// TIA Portal project "Project_Metrou" (V15.1)

(* hardware
DEVICE "S71500/ET200MP station_1"  S7-1500 station
   slot 0: "Rail_0"  Rack  6ES7 590-1***0-0AA0
   slot 1: "PLC_1"  CPU 1513-1 PN  6ES7 513-1AL02-0AB0  V2.6
      slot 3: "CPU display_1"  6ES7591-1AA00-0AA0
DEVICE "HMI_1"  KTP900 Basic PN
   slot 0: "HMI_1"  KTP900 Basic PN  6AV2 123-2JB03-0AX0  15.1.0.0
   slot 1: "HMI_RT_1"  KTP900 Basic PN  6AV2 123-2JB03-0AX0  15.1.0.0
   slot 5: "HMI_1.IE_CP_1"  PROFINET Interface  15.0.1.0
      slot 1: "PROFINET Interface_1"  PROFINET Interface
         slot 1: "Port_1"  Port
*)

// ===== PLC "PLC_1"  CPU 1513-1 PN =====

DATA_BLOCK "Alarme_scara"   // DB1
{ S7_Optimized_Access := 'TRUE' }
VERSION : 0.1
   VAR
      alarme_gather : Word;
      alarme_vect : Array[0..15] of Bool;
   END_VAR
BEGIN
END_DATA_BLOCK

DATA_BLOCK "Avarii"   // DB2
{ S7_Optimized_Access := 'TRUE' }
VERSION : 0.1
   VAR
      esd : Bool;
      esd_btn : Bool;
      reset_esd : Bool;
      avarie_s1 : Bool;
      avarie_s2 : Bool;
      avarie_p1 : Bool;
      avarie_p2 : Bool;
      reset_avarii : Bool;
   END_VAR
BEGIN
END_DATA_BLOCK

DATA_BLOCK "Alarme_poarta"   // DB3
{ S7_Optimized_Access := 'TRUE' }
VERSION : 0.1
   VAR
      alarme_gather : Word;
      alarme_vect : Array[0..15] of Bool;
   END_VAR
BEGIN
END_DATA_BLOCK

DATA_BLOCK "Scara1_DB"   // DB4
{ S7_Optimized_Access := 'TRUE' }
VERSION : 0.1
// stored: InstanceOfName Scara
"Scara"
BEGIN
END_DATA_BLOCK

DATA_BLOCK "Scara2_DB"   // DB5
{ S7_Optimized_Access := 'TRUE' }
VERSION : 0.1
// stored: InstanceOfName Scara
"Scara"
BEGIN
END_DATA_BLOCK

DATA_BLOCK "Variabile_scara1"   // DB6
{ S7_Optimized_Access := 'TRUE' }
VERSION : 0.1
   VAR
      curent_stea : Real;
      curent_triunghi : Real;
      senzor_presiune : Bool;
      porniire_stea : Bool;
      pornire_triunghi : Bool;
      start : Bool;
      stop : Bool;
      directie : Bool;
      sus : Bool;
      jos : Bool;
      reseteaza_directia : Bool;
      start_sus : Bool;
      start_jos : Bool;
      cartela_intr : Bool;
   END_VAR
BEGIN
END_DATA_BLOCK

DATA_BLOCK "Variabile_scara2"   // DB7
{ S7_Optimized_Access := 'TRUE' }
VERSION : 0.1
   VAR
      curent_stea : Real;
      curent_triunghi : Real;
      senzor_presiune : Bool;
      porniire_stea : Bool;
      pornire_triunghi : Bool;
      start : Bool;
      stop : Bool;
      directie : Bool;
      sus : Bool;
      jos : Bool;
      reseteaza_directia : Bool;
      start_sus : Bool;
      start_jos : Bool;
      cartela_intr : Bool;
   END_VAR
BEGIN
END_DATA_BLOCK

DATA_BLOCK "Poarta1_DB"   // DB9
{ S7_Optimized_Access := 'TRUE' }
VERSION : 0.1
// stored: InstanceOfName Poarta
"Poarta"
BEGIN
END_DATA_BLOCK

DATA_BLOCK "Poarta2_DB"   // DB10
{ S7_Optimized_Access := 'TRUE' }
VERSION : 0.1
// stored: InstanceOfName Poarta
"Poarta"
BEGIN
END_DATA_BLOCK

DATA_BLOCK "Variabile_poarta1"   // DB11
{ S7_Optimized_Access := 'TRUE' }
VERSION : 0.1
   VAR
      cartela : Bool;
      stop : Bool;
      start : Bool;
      permisiune_start : Bool;
      start_intrare : Bool;
      start_iesire : Bool;
      s1 : Bool;
      s2 : Bool;
      p_deschis : Bool;
      alarma : Bool;
   END_VAR
BEGIN
END_DATA_BLOCK

DATA_BLOCK "Variabile_poarta2"   // DB12
{ S7_Optimized_Access := 'TRUE' }
VERSION : 0.1
   VAR
      cartela : Bool;
      stop : Bool;
      start : Bool;
      permisiune_start : Bool;
      start_intrare : Bool;
      start_iesire : Bool;
      s1 : Bool;
      s2 : Bool;
      p_deschis : Bool;
      alarma : Bool;
   END_VAR
BEGIN
END_DATA_BLOCK

// folder: System blocks/Program resources

DATA_BLOCK "reset_esd"   // DB8
{ S7_Optimized_Access := 'TRUE' }
AUTHOR : Simatic
FAMILY : IEC
NAME : IEC_TMR
VERSION : 1.0
// stored: InstanceOfName IEC_TIMER
"IEC_TIMER"
BEGIN
END_DATA_BLOCK

// folder: (top level)

FUNCTION_BLOCK "Scara"   // FB1, LAD
{ S7_Optimized_Access := 'TRUE' }
VERSION : 0.1
   VAR_INPUT
      esd : Bool;
      curent_stea : Real;
      curent_triunghi : Real;
      avarie_scara : Bool;
   END_VAR
   VAR_OUTPUT
      stea : Bool;
      triunghi : Bool;
   END_VAR
   VAR_IN_OUT
      senzor_presiune : Bool;
      reseteaza_directia : Bool;
      stop : Bool;
      start : Bool;
      start_sus : Bool;
      start_jos : Bool;
   END_VAR
   VAR
      sus : Bool;
      jos : Bool;
      pornire_stea : Bool;
      pornire_triunghi : Bool;
      permisiune_pornire : Bool;
      permisie_repornire : Bool;
      timer_stop : TON_TIME;
      Motor : "Motor";
   END_VAR
BEGIN

REGION Network 1: da permisiuneade pornire la scara
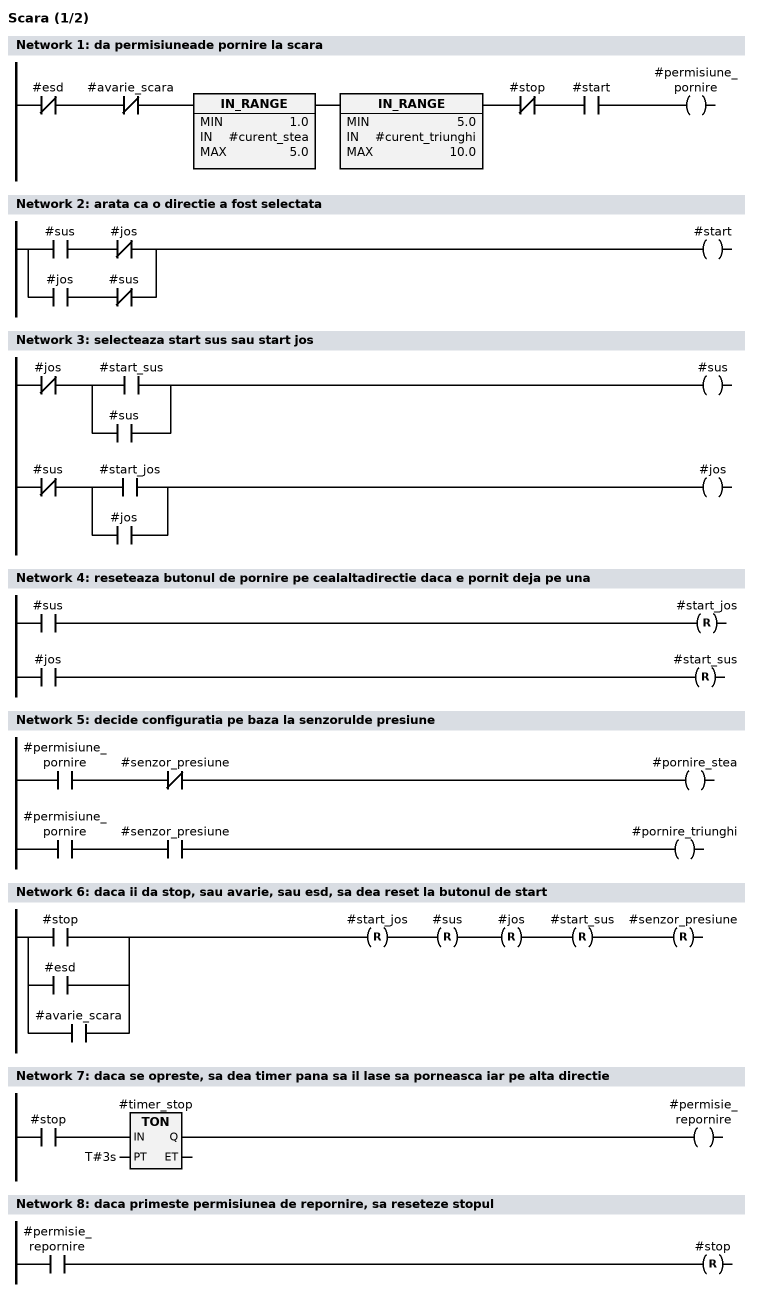
   RUNG wire#powerrail
      I_Contact( #esd )
      I_Contact( #avarie_scara )
      { S7_Templates := "SrcType := Real" } InRange(min := 1.0, in := #curent_stea, max := 5.0)
      { S7_Templates := "SrcType := Real" } InRange(min := 5.0, in := #curent_triunghi, max := 10.0)
      I_Contact( #stop )
      Contact( #start )
      Coil( #permisiune_pornire )
   END_RUNG
   // the same network as SCL:
   #permisiune_pornire := NOT #esd AND NOT #avarie_scara AND (1.0 <= #curent_stea) AND (#curent_stea <= 5.0) AND (5.0 <= #curent_triunghi) AND (#curent_triunghi <= 10.0) AND NOT #stop AND #start;
END_REGION

REGION Network 2: arata ca o directie a fost selectata
   RUNG wire#powerrail
      Contact( #sus )
      I_Contact( #jos )
      wire#w1
      Coil( #start )
   END_RUNG
   RUNG wire#powerrail
      Contact( #jos )
      I_Contact( #sus )
   END_RUNG wire#w1
   // the same network as SCL:
   #start := (#sus AND NOT #jos) OR (#jos AND NOT #sus);
END_REGION

REGION Network 3: selecteaza start sus sau start jos
   RUNG wire#powerrail
      I_Contact( #jos )
      wire#w1
      Contact( #start_sus )
      wire#w2
      Coil( #sus )
   END_RUNG
   RUNG wire#w1
      Contact( #sus )
   END_RUNG wire#w2
   RUNG wire#powerrail
      I_Contact( #sus )
      wire#w3
      Contact( #start_jos )
      wire#w4
      Coil( #jos )
   END_RUNG
   RUNG wire#w3
      Contact( #jos )
   END_RUNG wire#w4
   // the same network as SCL:
   #sus := NOT #jos AND (#start_sus OR #sus);
   #jos := NOT #sus AND (#start_jos OR #jos);
END_REGION

REGION Network 4: reseteaza butonul de pornire pe cealaltadirectie daca e pornit deja pe una
   RUNG wire#powerrail
      Contact( #sus )
      R_Coil( #start_jos )
   END_RUNG
   RUNG wire#powerrail
      Contact( #jos )
      R_Coil( #start_sus )
   END_RUNG
   // the same network as SCL:
   IF #sus THEN #start_jos := FALSE; END_IF;
   IF #jos THEN #start_sus := FALSE; END_IF;
END_REGION

REGION Network 5: decide configuratia pe baza la senzorulde presiune
   RUNG wire#powerrail
      Contact( #permisiune_pornire )
      I_Contact( #senzor_presiune )
      Coil( #pornire_stea )
   END_RUNG
   RUNG wire#powerrail
      Contact( #permisiune_pornire )
      Contact( #senzor_presiune )
      Coil( #pornire_triunghi )
   END_RUNG
   // the same network as SCL:
   #pornire_stea := #permisiune_pornire AND NOT #senzor_presiune;
   #pornire_triunghi := #permisiune_pornire AND #senzor_presiune;
END_REGION

REGION Network 6: daca ii da stop, sau avarie, sau esd, sa dea reset la butonul de start
   RUNG wire#powerrail
      Contact( #stop )
      wire#w1
      R_Coil( #start_jos )
      R_Coil( #sus )
      R_Coil( #jos )
      R_Coil( #start_sus )
      R_Coil( #senzor_presiune )
   END_RUNG
   RUNG wire#powerrail
      Contact( #esd )
   END_RUNG wire#w1
   RUNG wire#powerrail
      Contact( #avarie_scara )
   END_RUNG wire#w1
   // the same network as SCL:
   IF #stop OR #esd OR #avarie_scara THEN
       #start_jos := FALSE;
       #sus := FALSE;
       #jos := FALSE;
       #start_sus := FALSE;
       #senzor_presiune := FALSE;
   END_IF;
END_REGION

REGION Network 7: daca se opreste, sa dea timer pana sa il lase sa porneasca iar pe alta directie
   #timer_stop(IN := #stop, PT := T#3s);   // TON
   #permisie_repornire := #timer_stop.Q;
END_REGION

REGION Network 8: daca primeste permisiunea de repornire, sa reseteze stopul
   RUNG wire#powerrail
      Contact( #permisie_repornire )
      R_Coil( #stop )
   END_RUNG
   // the same network as SCL:
   IF #permisie_repornire THEN #stop := FALSE; END_IF;
END_REGION

REGION Network 9: functia de motor a scarii
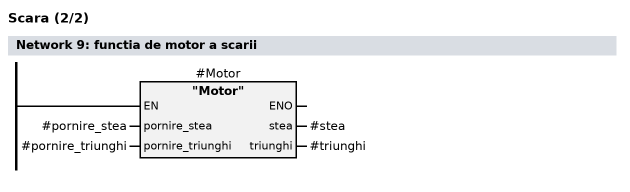
   RUNG wire#powerrail
      #Motor(pornire_stea := #pornire_stea, pornire_triunghi := #pornire_triunghi, stea => #stea, triunghi => #triunghi)
   END_RUNG
   // the same network as SCL:
   #Motor(pornire_stea := #pornire_stea,   // "Motor"
          pornire_triunghi := #pornire_triunghi,
          stea => #stea,
          triunghi => #triunghi);
END_REGION
END_FUNCTION_BLOCK

FUNCTION_BLOCK "Motor"   // FB2, LAD
{ S7_Optimized_Access := 'TRUE' }
VERSION : 0.1
   VAR_INPUT
      pornire_stea : Bool;
      pornire_triunghi : Bool;
   END_VAR
   VAR_OUTPUT
      stea : Bool;
      triunghi : Bool;
   END_VAR
BEGIN

REGION Network 1: daca primeste plecare pe stea, sa o activeze
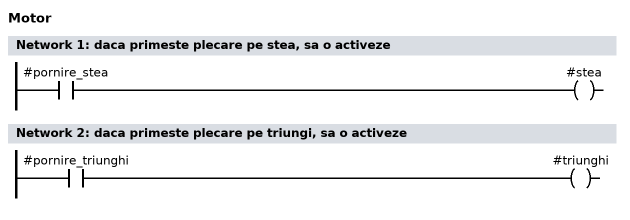
   RUNG wire#powerrail
      Contact( #pornire_stea )
      Coil( #stea )
   END_RUNG
   // the same network as SCL:
   #stea := #pornire_stea;
END_REGION

REGION Network 2: daca primeste plecare pe triungi, sa o activeze
   RUNG wire#powerrail
      Contact( #pornire_triunghi )
      Coil( #triunghi )
   END_RUNG
   // the same network as SCL:
   #triunghi := #pornire_triunghi;
END_REGION
END_FUNCTION_BLOCK

FUNCTION_BLOCK "Poarta"   // FB3, LAD
{ S7_Optimized_Access := 'TRUE' }
VERSION : 0.1
   VAR_INPUT
      esd : Bool;
      avarie_poarta : Bool;
   END_VAR
   VAR_OUTPUT
      poarta_deschisa : Bool;
      alarma : Bool;
   END_VAR
   VAR_IN_OUT
      senzor1 : Bool;
      senzor2 : Bool;
      cartela : Bool;
      stop : Bool;
      start : Bool;
      permisiune_start : Bool;
      start_intrare : Bool;
      start_iesire : Bool;
      cartela_introdusa : Bool;
   END_VAR
   VAR
      terminat1 : Bool;
      terminat2 : Bool;
      intrare : Bool;
      s1_intrare : Bool;
      s1_iesire : Bool;
      s2_intrare : Bool;
      s2_iesire : Bool;
      iesire : Bool;
      reset_stop : TON_TIME;
      Iesire_metrou_Instance : "Iesire_metrou";
      Intrare_metrou_Instance : "Intrare_metrou";
   END_VAR
BEGIN

REGION Network 1: porneste poarta
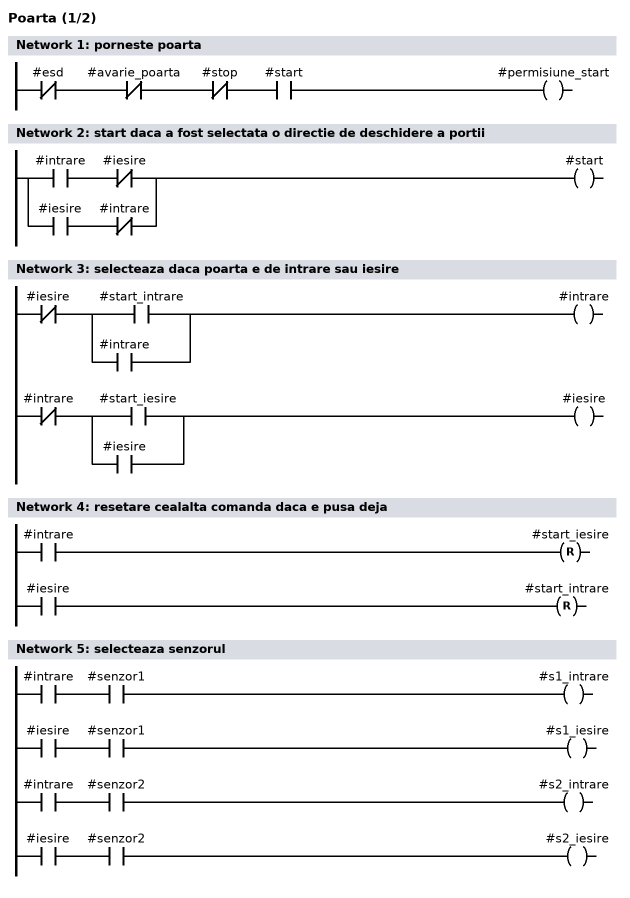
   RUNG wire#powerrail
      I_Contact( #esd )
      I_Contact( #avarie_poarta )
      I_Contact( #stop )
      Contact( #start )
      Coil( #permisiune_start )
   END_RUNG
   // the same network as SCL:
   #permisiune_start := NOT #esd AND NOT #avarie_poarta AND NOT #stop AND #start;
END_REGION

REGION Network 2: start daca a fost selectata o directie de deschidere a portii
   RUNG wire#powerrail
      Contact( #intrare )
      I_Contact( #iesire )
      wire#w1
      Coil( #start )
   END_RUNG
   RUNG wire#powerrail
      Contact( #iesire )
      I_Contact( #intrare )
   END_RUNG wire#w1
   // the same network as SCL:
   #start := (#intrare AND NOT #iesire) OR (#iesire AND NOT #intrare);
END_REGION

REGION Network 3: selecteaza daca poarta e de intrare sau iesire
   RUNG wire#powerrail
      I_Contact( #iesire )
      wire#w1
      Contact( #start_intrare )
      wire#w2
      Coil( #intrare )
   END_RUNG
   RUNG wire#w1
      Contact( #intrare )
   END_RUNG wire#w2
   RUNG wire#powerrail
      I_Contact( #intrare )
      wire#w3
      Contact( #start_iesire )
      wire#w4
      Coil( #iesire )
   END_RUNG
   RUNG wire#w3
      Contact( #iesire )
   END_RUNG wire#w4
   // the same network as SCL:
   #intrare := NOT #iesire AND (#start_intrare OR #intrare);
   #iesire := NOT #intrare AND (#start_iesire OR #iesire);
END_REGION

REGION Network 4: resetare cealalta comanda daca e pusa deja
   RUNG wire#powerrail
      Contact( #intrare )
      R_Coil( #start_iesire )
   END_RUNG
   RUNG wire#powerrail
      Contact( #iesire )
      R_Coil( #start_intrare )
   END_RUNG
   // the same network as SCL:
   IF #intrare THEN #start_iesire := FALSE; END_IF;
   IF #iesire THEN #start_intrare := FALSE; END_IF;
END_REGION

REGION Network 5: selecteaza senzorul
   RUNG wire#powerrail
      Contact( #intrare )
      Contact( #senzor1 )
      Coil( #s1_intrare )
   END_RUNG
   RUNG wire#powerrail
      Contact( #iesire )
      Contact( #senzor1 )
      Coil( #s1_iesire )
   END_RUNG
   RUNG wire#powerrail
      Contact( #intrare )
      Contact( #senzor2 )
      Coil( #s2_intrare )
   END_RUNG
   RUNG wire#powerrail
      Contact( #iesire )
      Contact( #senzor2 )
      Coil( #s2_iesire )
   END_RUNG
   // the same network as SCL:
   #s1_intrare := #intrare AND #senzor1;
   #s1_iesire := #iesire AND #senzor1;
   #s2_intrare := #intrare AND #senzor2;
   #s2_iesire := #iesire AND #senzor2;
END_REGION

REGION Network 6: functie intrare/iesire
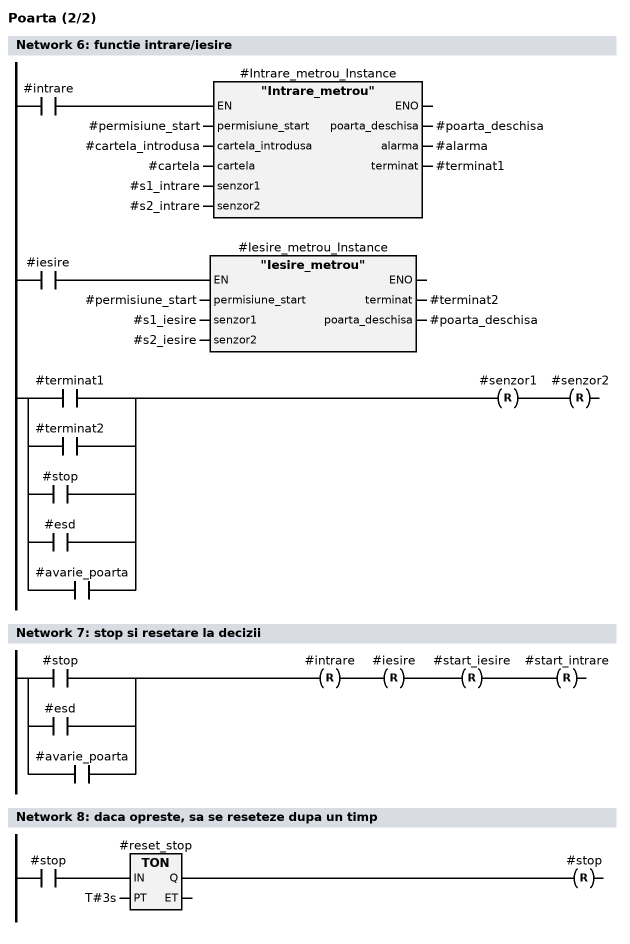
   RUNG wire#powerrail
      Contact( #intrare )
      #Intrare_metrou_Instance(permisiune_start := #permisiune_start, cartela_introdusa := #cartela_introdusa, cartela := #cartela, senzor1 := #s1_intrare, senzor2 := #s2_intrare, poarta_deschisa => #poarta_deschisa, alarma => #alarma, terminat => #terminat1)
   END_RUNG
   RUNG wire#powerrail
      Contact( #iesire )
      #Iesire_metrou_Instance(permisiune_start := #permisiune_start, senzor1 := #s1_iesire, senzor2 := #s2_iesire, terminat => #terminat2, poarta_deschisa => #poarta_deschisa)
   END_RUNG
   RUNG wire#powerrail
      Contact( #terminat1 )
      wire#w1
      R_Coil( #senzor1 )
      R_Coil( #senzor2 )
   END_RUNG
   RUNG wire#powerrail
      Contact( #terminat2 )
   END_RUNG wire#w1
   RUNG wire#powerrail
      Contact( #stop )
   END_RUNG wire#w1
   RUNG wire#powerrail
      Contact( #esd )
   END_RUNG wire#w1
   RUNG wire#powerrail
      Contact( #avarie_poarta )
   END_RUNG wire#w1
   // the same network as SCL:
   IF #intrare THEN
       #Intrare_metrou_Instance(permisiune_start := #permisiune_start,   // "Intrare_metrou"
                               cartela_introdusa := #cartela_introdusa,
                               cartela := #cartela,
                               senzor1 := #s1_intrare,
                               senzor2 := #s2_intrare,
                               poarta_deschisa => #poarta_deschisa,
                               alarma => #alarma,
                               terminat => #terminat1);
   END_IF;
   IF #iesire THEN
       #Iesire_metrou_Instance(permisiune_start := #permisiune_start,   // "Iesire_metrou"
                               senzor1 := #s1_iesire,
                               senzor2 := #s2_iesire,
                               terminat => #terminat2,
                               poarta_deschisa => #poarta_deschisa);
   END_IF;
   IF #terminat1 OR #terminat2 OR #stop OR #esd OR #avarie_poarta THEN
       #senzor1 := FALSE;
       #senzor2 := FALSE;
   END_IF;
END_REGION

REGION Network 7: stop si resetare la decizii
   RUNG wire#powerrail
      Contact( #stop )
      wire#w1
      R_Coil( #intrare )
      R_Coil( #iesire )
      R_Coil( #start_iesire )
      R_Coil( #start_intrare )
   END_RUNG
   RUNG wire#powerrail
      Contact( #esd )
   END_RUNG wire#w1
   RUNG wire#powerrail
      Contact( #avarie_poarta )
   END_RUNG wire#w1
   // the same network as SCL:
   IF #stop OR #esd OR #avarie_poarta THEN
       #intrare := FALSE;
       #iesire := FALSE;
       #start_iesire := FALSE;
       #start_intrare := FALSE;
   END_IF;
END_REGION

REGION Network 8: daca opreste, sa se reseteze dupa un timp
   #reset_stop(IN := #stop, PT := T#3s);   // TON
   IF #reset_stop.Q THEN #stop := FALSE; END_IF;
END_REGION
END_FUNCTION_BLOCK

FUNCTION_BLOCK "Intrare_metrou"   // FB4, LAD
{ S7_Optimized_Access := 'TRUE' }
VERSION : 0.1
   VAR_INPUT
      permisiune_start : Bool;
   END_VAR
   VAR_OUTPUT
      poarta_deschisa : Bool;
      alarma : Bool;
      terminat : Bool;
   END_VAR
   VAR_IN_OUT
      cartela_introdusa : Bool;
      cartela : Bool;
      senzor1 : Bool;
      senzor2 : Bool;
   END_VAR
   VAR
      timer_alarma : TON_TIME;
   END_VAR
BEGIN

REGION Network 1
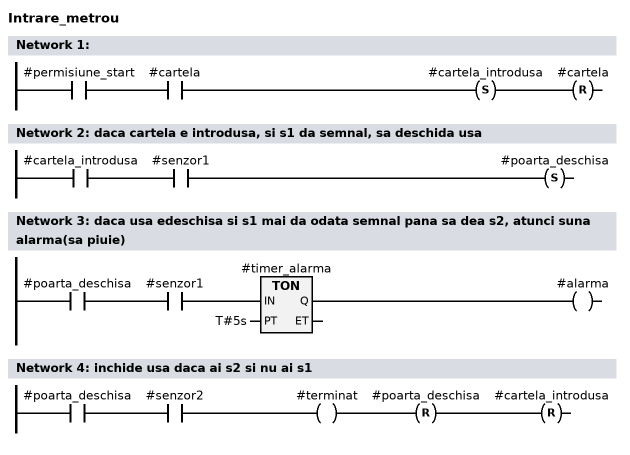
   RUNG wire#powerrail
      Contact( #permisiune_start )
      Contact( #cartela )
      S_Coil( #cartela_introdusa )
      R_Coil( #cartela )
   END_RUNG
   // the same network as SCL:
   IF #permisiune_start AND #cartela THEN
       #cartela_introdusa := TRUE;
       #cartela := FALSE;
   END_IF;
END_REGION

REGION Network 2: daca cartela e introdusa, si s1 da semnal, sa deschida usa
   RUNG wire#powerrail
      Contact( #cartela_introdusa )
      Contact( #senzor1 )
      S_Coil( #poarta_deschisa )
   END_RUNG
   // the same network as SCL:
   IF #cartela_introdusa AND #senzor1 THEN #poarta_deschisa := TRUE; END_IF;
END_REGION

REGION Network 3: daca usa edeschisa si s1 mai da odata semnal pana sa dea s2, atunci suna alarma(sa piuie)
   #timer_alarma(IN := #poarta_deschisa AND #senzor1, PT := T#5s);   // TON
   #alarma := #timer_alarma.Q;
END_REGION

REGION Network 4: inchide usa daca ai s2 si nu ai s1
   RUNG wire#powerrail
      Contact( #poarta_deschisa )
      Contact( #senzor2 )
      Coil( #terminat )
      R_Coil( #poarta_deschisa )
      R_Coil( #cartela_introdusa )
   END_RUNG
   // the same network as SCL:
   #terminat := #poarta_deschisa AND #senzor2;
   IF #terminat THEN
       #poarta_deschisa := FALSE;
       #cartela_introdusa := FALSE;
   END_IF;
END_REGION
END_FUNCTION_BLOCK

FUNCTION_BLOCK "Iesire_metrou"   // FB5, LAD
{ S7_Optimized_Access := 'TRUE' }
VERSION : 0.1
   VAR_INPUT
      permisiune_start : Bool;
   END_VAR
   VAR_OUTPUT
      terminat : Bool;
      poarta_deschisa : Bool;
   END_VAR
   VAR_IN_OUT
      senzor1 : Bool;
      senzor2 : Bool;
   END_VAR
BEGIN

REGION Network 1: deschide poarta daca senzor1 da semnal
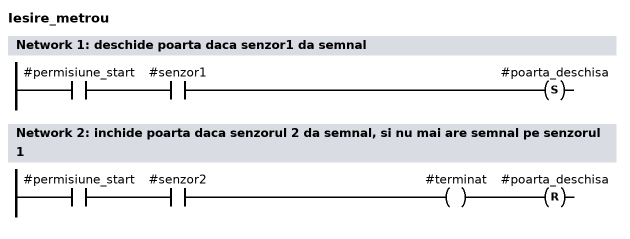
   RUNG wire#powerrail
      Contact( #permisiune_start )
      Contact( #senzor1 )
      S_Coil( #poarta_deschisa )
   END_RUNG
   // the same network as SCL:
   IF #permisiune_start AND #senzor1 THEN #poarta_deschisa := TRUE; END_IF;
END_REGION

REGION Network 2: inchide poarta daca senzorul 2 da semnal, si nu mai are semnal pe senzorul 1
   RUNG wire#powerrail
      Contact( #permisiune_start )
      Contact( #senzor2 )
      Coil( #terminat )
      R_Coil( #poarta_deschisa )
   END_RUNG
   // the same network as SCL:
   #terminat := #permisiune_start AND #senzor2;
   IF #terminat THEN #poarta_deschisa := FALSE; END_IF;
END_REGION
END_FUNCTION_BLOCK

ORGANIZATION_BLOCK "Main"   // OB1, LAD, ProgramCycle
TITLE = "Main Program Sweep (Cycle)"
{ S7_Optimized_Access := 'TRUE' }
VERSION : 0.1
   VAR_INPUT
      Initial_Call : Bool;   // Initial call of this OB
      Remanence : Bool;   // =True, if remanent data are available
   END_VAR
   VAR_TEMP   // added for the SCL form of the ladder/FBD networks
      _w1 : Bool;
      _w2 : Bool;
      _w3 : Bool;
      _w4 : Bool;
   END_VAR
BEGIN

REGION Network 1: scara 1
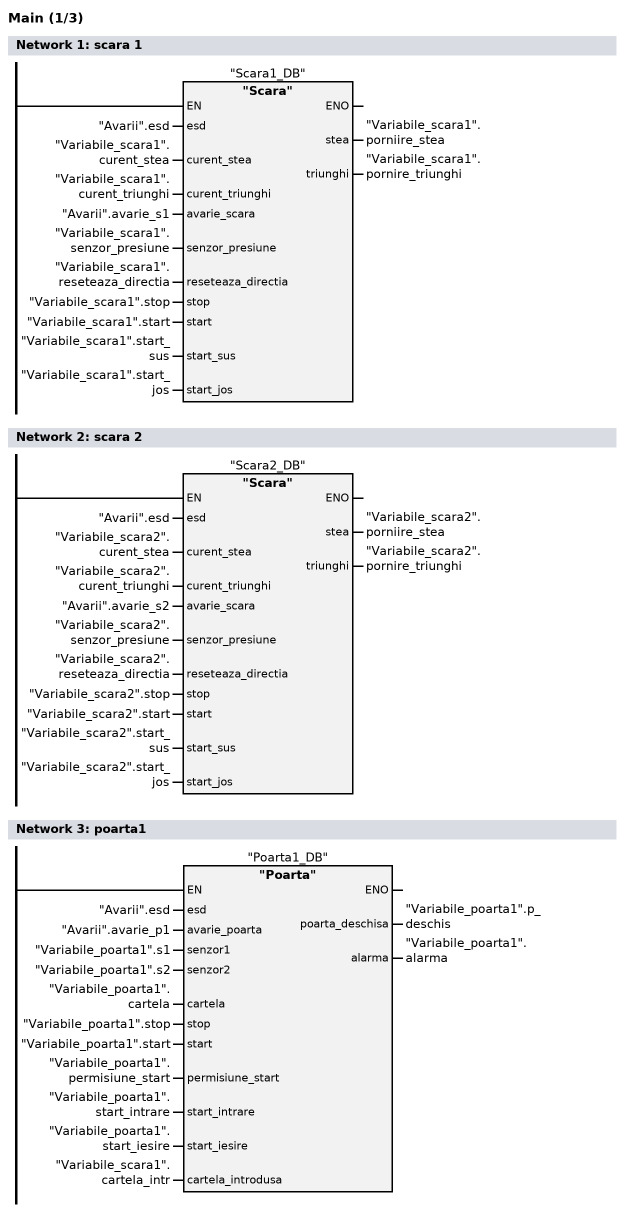
   RUNG wire#powerrail
      "Scara1_DB"(esd := "Avarii".esd, curent_stea := "Variabile_scara1".curent_stea, curent_triunghi := "Variabile_scara1".curent_triunghi, avarie_scara := "Avarii".avarie_s1, senzor_presiune := "Variabile_scara1".senzor_presiune, reseteaza_directia := "Variabile_scara1".reseteaza_directia, stop := "Variabile_scara1".stop, start := "Variabile_scara1".start, start_sus := "Variabile_scara1".start_sus, start_jos := "Variabile_scara1".start_jos, stea => "Variabile_scara1".porniire_stea, triunghi => "Variabile_scara1".pornire_triunghi)
   END_RUNG
   // the same network as SCL:
   "Scara1_DB"(esd := "Avarii".esd,   // "Scara"
               curent_stea := "Variabile_scara1".curent_stea,
               curent_triunghi := "Variabile_scara1".curent_triunghi,
               avarie_scara := "Avarii".avarie_s1,
               senzor_presiune := "Variabile_scara1".senzor_presiune,
               reseteaza_directia := "Variabile_scara1".reseteaza_directia,
               stop := "Variabile_scara1".stop,
               start := "Variabile_scara1".start,
               start_sus := "Variabile_scara1".start_sus,
               start_jos := "Variabile_scara1".start_jos,
               stea => "Variabile_scara1".porniire_stea,
               triunghi => "Variabile_scara1".pornire_triunghi);
END_REGION

REGION Network 2: scara 2
   RUNG wire#powerrail
      "Scara2_DB"(esd := "Avarii".esd, curent_stea := "Variabile_scara2".curent_stea, curent_triunghi := "Variabile_scara2".curent_triunghi, avarie_scara := "Avarii".avarie_s2, senzor_presiune := "Variabile_scara2".senzor_presiune, reseteaza_directia := "Variabile_scara2".reseteaza_directia, stop := "Variabile_scara2".stop, start := "Variabile_scara2".start, start_sus := "Variabile_scara2".start_sus, start_jos := "Variabile_scara2".start_jos, stea => "Variabile_scara2".porniire_stea, triunghi => "Variabile_scara2".pornire_triunghi)
   END_RUNG
   // the same network as SCL:
   "Scara2_DB"(esd := "Avarii".esd,   // "Scara"
               curent_stea := "Variabile_scara2".curent_stea,
               curent_triunghi := "Variabile_scara2".curent_triunghi,
               avarie_scara := "Avarii".avarie_s2,
               senzor_presiune := "Variabile_scara2".senzor_presiune,
               reseteaza_directia := "Variabile_scara2".reseteaza_directia,
               stop := "Variabile_scara2".stop,
               start := "Variabile_scara2".start,
               start_sus := "Variabile_scara2".start_sus,
               start_jos := "Variabile_scara2".start_jos,
               stea => "Variabile_scara2".porniire_stea,
               triunghi => "Variabile_scara2".pornire_triunghi);
END_REGION

REGION Network 3: poarta1
   RUNG wire#powerrail
      "Poarta1_DB"(esd := "Avarii".esd, avarie_poarta := "Avarii".avarie_p1, senzor1 := "Variabile_poarta1".s1, senzor2 := "Variabile_poarta1".s2, cartela := "Variabile_poarta1".cartela, stop := "Variabile_poarta1".stop, start := "Variabile_poarta1".start, permisiune_start := "Variabile_poarta1".permisiune_start, start_intrare := "Variabile_poarta1".start_intrare, start_iesire := "Variabile_poarta1".start_iesire, cartela_introdusa := "Variabile_scara1".cartela_intr, poarta_deschisa => "Variabile_poarta1".p_deschis, alarma => "Variabile_poarta1".alarma)
   END_RUNG
   // the same network as SCL:
   "Poarta1_DB"(esd := "Avarii".esd,   // "Poarta"
                avarie_poarta := "Avarii".avarie_p1,
                senzor1 := "Variabile_poarta1".s1,
                senzor2 := "Variabile_poarta1".s2,
                cartela := "Variabile_poarta1".cartela,
                stop := "Variabile_poarta1".stop,
                start := "Variabile_poarta1".start,
                permisiune_start := "Variabile_poarta1".permisiune_start,
                start_intrare := "Variabile_poarta1".start_intrare,
                start_iesire := "Variabile_poarta1".start_iesire,
                cartela_introdusa := "Variabile_scara1".cartela_intr,
                poarta_deschisa => "Variabile_poarta1".p_deschis,
                alarma => "Variabile_poarta1".alarma);
END_REGION

REGION Network 4: poarta2
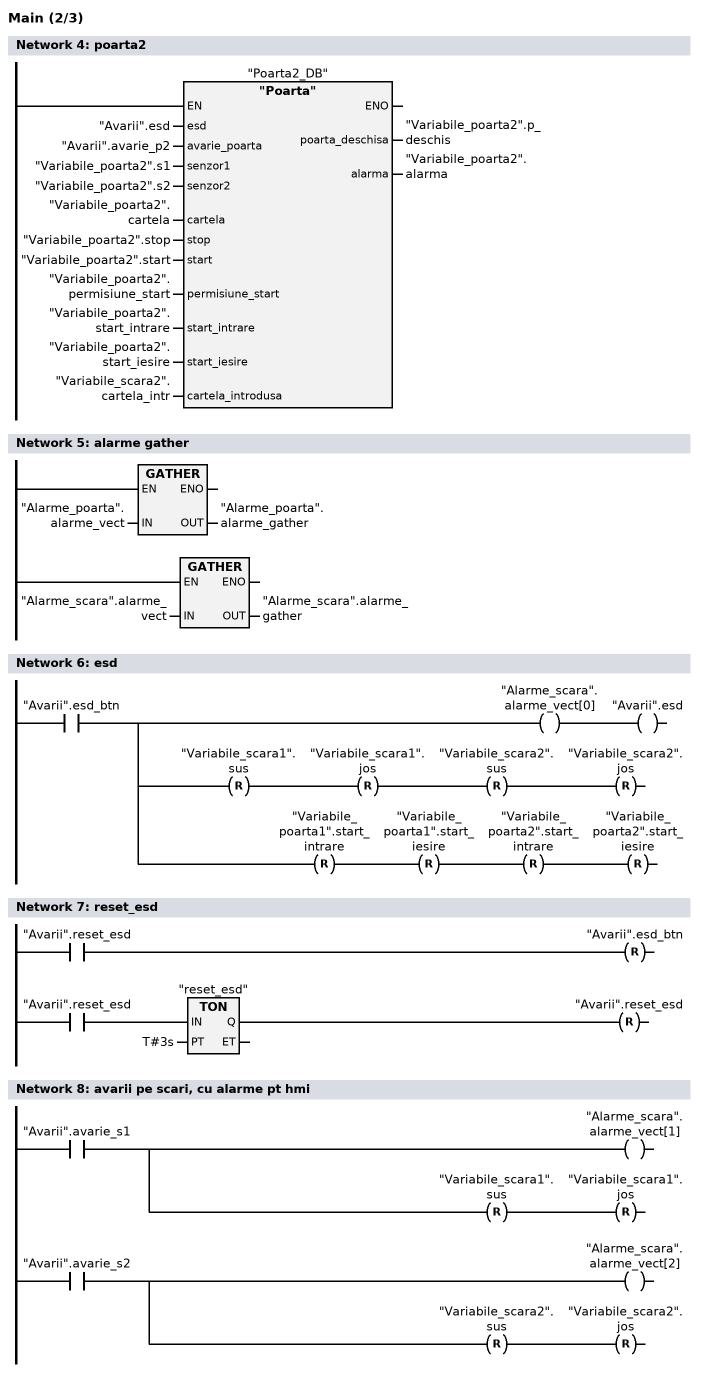
   RUNG wire#powerrail
      "Poarta2_DB"(esd := "Avarii".esd, avarie_poarta := "Avarii".avarie_p2, senzor1 := "Variabile_poarta2".s1, senzor2 := "Variabile_poarta2".s2, cartela := "Variabile_poarta2".cartela, stop := "Variabile_poarta2".stop, start := "Variabile_poarta2".start, permisiune_start := "Variabile_poarta2".permisiune_start, start_intrare := "Variabile_poarta2".start_intrare, start_iesire := "Variabile_poarta2".start_iesire, cartela_introdusa := "Variabile_scara2".cartela_intr, poarta_deschisa => "Variabile_poarta2".p_deschis, alarma => "Variabile_poarta2".alarma)
   END_RUNG
   // the same network as SCL:
   "Poarta2_DB"(esd := "Avarii".esd,   // "Poarta"
                avarie_poarta := "Avarii".avarie_p2,
                senzor1 := "Variabile_poarta2".s1,
                senzor2 := "Variabile_poarta2".s2,
                cartela := "Variabile_poarta2".cartela,
                stop := "Variabile_poarta2".stop,
                start := "Variabile_poarta2".start,
                permisiune_start := "Variabile_poarta2".permisiune_start,
                start_intrare := "Variabile_poarta2".start_intrare,
                start_iesire := "Variabile_poarta2".start_iesire,
                cartela_introdusa := "Variabile_scara2".cartela_intr,
                poarta_deschisa => "Variabile_poarta2".p_deschis,
                alarma => "Variabile_poarta2".alarma);
END_REGION

REGION Network 5: alarme gather
   GATHER(IN := "Alarme_poarta".alarme_vect, OUT => "Alarme_poarta".alarme_gather);
   GATHER(IN := "Alarme_scara".alarme_vect, OUT => "Alarme_scara".alarme_gather);
END_REGION

REGION Network 6: esd
   RUNG wire#powerrail
      Contact( "Avarii".esd_btn )
      wire#w1
      Coil( "Alarme_scara".alarme_vect[0] )
      Coil( "Avarii".esd )
   END_RUNG
   RUNG wire#w1
      R_Coil( "Variabile_scara1".sus )
      R_Coil( "Variabile_scara1".jos )
      R_Coil( "Variabile_scara2".sus )
      R_Coil( "Variabile_scara2".jos )
   END_RUNG
   RUNG wire#w1
      R_Coil( "Variabile_poarta1".start_intrare )
      R_Coil( "Variabile_poarta1".start_iesire )
      R_Coil( "Variabile_poarta2".start_intrare )
      R_Coil( "Variabile_poarta2".start_iesire )
   END_RUNG
   // the same network as SCL:
   "Alarme_scara".alarme_vect[0] := "Avarii".esd_btn;
   "Avarii".esd := "Avarii".esd_btn;
   IF "Avarii".esd_btn THEN
       "Variabile_scara1".sus := FALSE;
       "Variabile_scara1".jos := FALSE;
       "Variabile_scara2".sus := FALSE;
       "Variabile_scara2".jos := FALSE;
       "Variabile_poarta1".start_intrare := FALSE;
       "Variabile_poarta1".start_iesire := FALSE;
       "Variabile_poarta2".start_intrare := FALSE;
       "Variabile_poarta2".start_iesire := FALSE;
   END_IF;
END_REGION

REGION Network 7: reset_esd
   IF "Avarii".reset_esd THEN "Avarii".esd_btn := FALSE; END_IF;
   "reset_esd".TON(IN := "Avarii".reset_esd, PT := T#3s);
   IF "reset_esd".Q THEN "Avarii".reset_esd := FALSE; END_IF;
END_REGION

REGION Network 8: avarii pe scari, cu alarme pt hmi
   RUNG wire#powerrail
      Contact( "Avarii".avarie_s1 )
      wire#w1
      Coil( "Alarme_scara".alarme_vect[1] )
   END_RUNG
   RUNG wire#w1
      R_Coil( "Variabile_scara1".sus )
      R_Coil( "Variabile_scara1".jos )
   END_RUNG
   RUNG wire#powerrail
      Contact( "Avarii".avarie_s2 )
      wire#w2
      Coil( "Alarme_scara".alarme_vect[2] )
   END_RUNG
   RUNG wire#w2
      R_Coil( "Variabile_scara2".sus )
      R_Coil( "Variabile_scara2".jos )
   END_RUNG
   // the same network as SCL:
   "Alarme_scara".alarme_vect[1] := "Avarii".avarie_s1;
   IF "Avarii".avarie_s1 THEN
       "Variabile_scara1".sus := FALSE;
       "Variabile_scara1".jos := FALSE;
   END_IF;
   "Alarme_scara".alarme_vect[2] := "Avarii".avarie_s2;
   IF "Avarii".avarie_s2 THEN
       "Variabile_scara2".sus := FALSE;
       "Variabile_scara2".jos := FALSE;
   END_IF;
END_REGION

REGION Network 9: reset la avarii
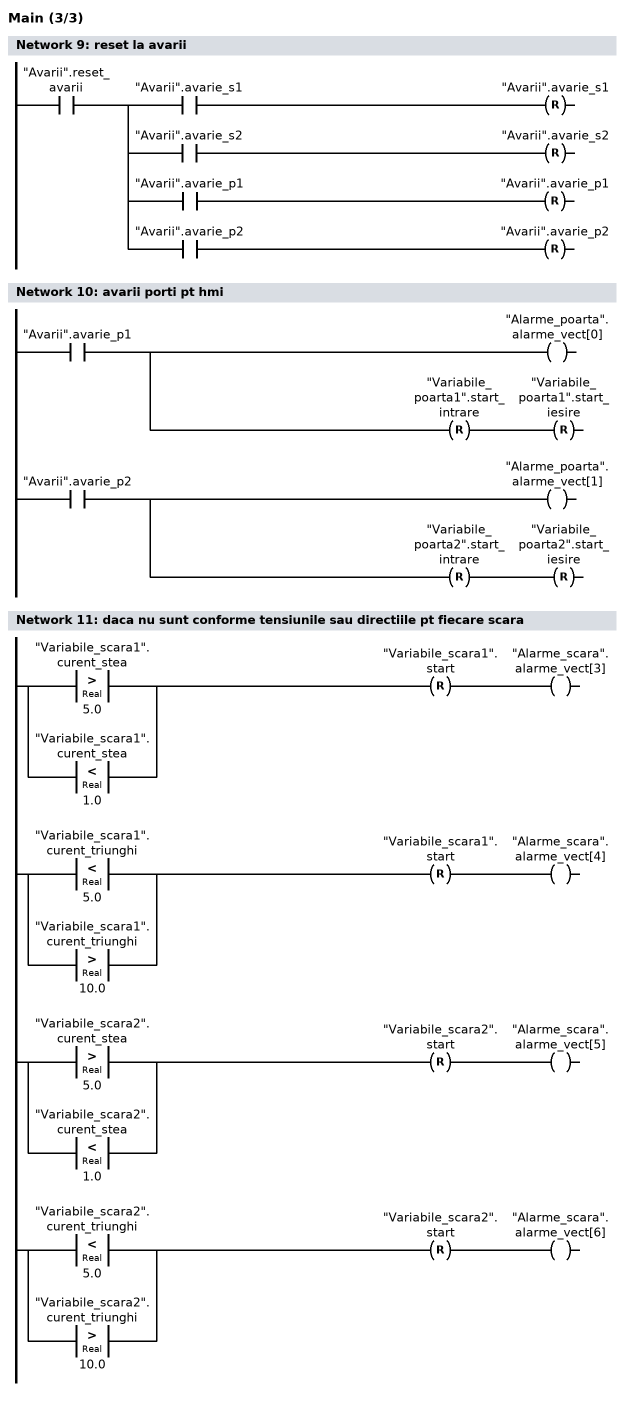
   RUNG wire#powerrail
      Contact( "Avarii".reset_avarii )
      wire#w1
      Contact( "Avarii".avarie_s1 )
      R_Coil( "Avarii".avarie_s1 )
   END_RUNG
   RUNG wire#w1
      Contact( "Avarii".avarie_s2 )
      R_Coil( "Avarii".avarie_s2 )
   END_RUNG
   RUNG wire#w1
      Contact( "Avarii".avarie_p1 )
      R_Coil( "Avarii".avarie_p1 )
   END_RUNG
   RUNG wire#w1
      Contact( "Avarii".avarie_p2 )
      R_Coil( "Avarii".avarie_p2 )
   END_RUNG
   // the same network as SCL:
   IF "Avarii".reset_avarii AND "Avarii".avarie_s1 THEN "Avarii".avarie_s1 := FALSE; END_IF;
   IF "Avarii".reset_avarii AND "Avarii".avarie_s2 THEN "Avarii".avarie_s2 := FALSE; END_IF;
   IF "Avarii".reset_avarii AND "Avarii".avarie_p1 THEN "Avarii".avarie_p1 := FALSE; END_IF;
   IF "Avarii".reset_avarii AND "Avarii".avarie_p2 THEN "Avarii".avarie_p2 := FALSE; END_IF;
END_REGION

REGION Network 10: avarii porti pt hmi
   RUNG wire#powerrail
      Contact( "Avarii".avarie_p1 )
      wire#w1
      Coil( "Alarme_poarta".alarme_vect[0] )
   END_RUNG
   RUNG wire#w1
      R_Coil( "Variabile_poarta1".start_intrare )
      R_Coil( "Variabile_poarta1".start_iesire )
   END_RUNG
   RUNG wire#powerrail
      Contact( "Avarii".avarie_p2 )
      wire#w2
      Coil( "Alarme_poarta".alarme_vect[1] )
   END_RUNG
   RUNG wire#w2
      R_Coil( "Variabile_poarta2".start_intrare )
      R_Coil( "Variabile_poarta2".start_iesire )
   END_RUNG
   // the same network as SCL:
   "Alarme_poarta".alarme_vect[0] := "Avarii".avarie_p1;
   IF "Avarii".avarie_p1 THEN
       "Variabile_poarta1".start_intrare := FALSE;
       "Variabile_poarta1".start_iesire := FALSE;
   END_IF;
   "Alarme_poarta".alarme_vect[1] := "Avarii".avarie_p2;
   IF "Avarii".avarie_p2 THEN
       "Variabile_poarta2".start_intrare := FALSE;
       "Variabile_poarta2".start_iesire := FALSE;
   END_IF;
END_REGION

REGION Network 11: daca nu sunt conforme tensiunile sau directiile pt fiecare scara
   RUNG wire#powerrail
      { S7_Templates := "SrcType := Real" } GT_Contact(in1 := "Variabile_scara1".curent_stea, in2 := 5.0)
      wire#w1
      R_Coil( "Variabile_scara1".start )
      Coil( "Alarme_scara".alarme_vect[3] )
   END_RUNG
   RUNG wire#powerrail
      { S7_Templates := "SrcType := Real" } LT_Contact(in1 := "Variabile_scara1".curent_stea, in2 := 1.0)
   END_RUNG wire#w1
   RUNG wire#powerrail
      { S7_Templates := "SrcType := Real" } LT_Contact(in1 := "Variabile_scara1".curent_triunghi, in2 := 5.0)
      wire#w2
      R_Coil( "Variabile_scara1".start )
      Coil( "Alarme_scara".alarme_vect[4] )
   END_RUNG
   RUNG wire#powerrail
      { S7_Templates := "SrcType := Real" } GT_Contact(in1 := "Variabile_scara1".curent_triunghi, in2 := 10.0)
   END_RUNG wire#w2
   RUNG wire#powerrail
      { S7_Templates := "SrcType := Real" } GT_Contact(in1 := "Variabile_scara2".curent_stea, in2 := 5.0)
      wire#w3
      R_Coil( "Variabile_scara2".start )
      Coil( "Alarme_scara".alarme_vect[5] )
   END_RUNG
   RUNG wire#powerrail
      { S7_Templates := "SrcType := Real" } LT_Contact(in1 := "Variabile_scara2".curent_stea, in2 := 1.0)
   END_RUNG wire#w3
   RUNG wire#powerrail
      { S7_Templates := "SrcType := Real" } LT_Contact(in1 := "Variabile_scara2".curent_triunghi, in2 := 5.0)
      wire#w4
      R_Coil( "Variabile_scara2".start )
      Coil( "Alarme_scara".alarme_vect[6] )
   END_RUNG
   RUNG wire#powerrail
      { S7_Templates := "SrcType := Real" } GT_Contact(in1 := "Variabile_scara2".curent_triunghi, in2 := 10.0)
   END_RUNG wire#w4
   // the same network as SCL:
   #_w1 := ("Variabile_scara1".curent_stea > 5.0) OR ("Variabile_scara1".curent_stea < 1.0);
   IF #_w1 THEN "Variabile_scara1".start := FALSE; END_IF;
   "Alarme_scara".alarme_vect[3] := #_w1;
   #_w2 := ("Variabile_scara1".curent_triunghi < 5.0) OR ("Variabile_scara1".curent_triunghi > 10.0);
   IF #_w2 THEN "Variabile_scara1".start := FALSE; END_IF;
   "Alarme_scara".alarme_vect[4] := #_w2;
   #_w3 := ("Variabile_scara2".curent_stea > 5.0) OR ("Variabile_scara2".curent_stea < 1.0);
   IF #_w3 THEN "Variabile_scara2".start := FALSE; END_IF;
   "Alarme_scara".alarme_vect[5] := #_w3;
   #_w4 := ("Variabile_scara2".curent_triunghi < 5.0) OR ("Variabile_scara2".curent_triunghi > 10.0);
   IF #_w4 THEN "Variabile_scara2".start := FALSE; END_IF;
   "Alarme_scara".alarme_vect[6] := #_w4;
END_REGION
END_ORGANIZATION_BLOCK

(* ===== HMI "HMI_RT_1" =====
system functions are stored by id; their names below are inferred from use
connection "HMI_Connection_1": ETHERNET, SMART_S7_1500_OMS

HMI tags "Default tag table"
   "Tag_ScreenNumber" : UInt, internal
   "Alarme_scara_alarme_gather" : Word = PLC Alarme_scara.alarme_gather, 1 s
   "Alarme_poarta_alarme_gather" : Word = PLC Alarme_poarta.alarme_gather, 1 s
   "Variabile_scara1_curent_triunghi" : Real = PLC Variabile_scara1.curent_triunghi, 1 s
   "Variabile_scara1_curent_stea" : Real = PLC Variabile_scara1.curent_stea, 1 s
   "Avarii_esd" : Bool = PLC Avarii.esd, 1 s
   "Avarii_esd_btn" : Bool = PLC Avarii.esd_btn, 1 s
   "Avarii_reset_esd" : Bool = PLC Avarii.reset_esd, 1 s
   "Avarii_avarie_s1" : Bool = PLC Avarii.avarie_s1, 1 s
   "Avarii_avarie_s2" : Bool = PLC Avarii.avarie_s2, 1 s
   "Avarii_avarie_p1" : Bool = PLC Avarii.avarie_p1, 1 s
   "Avarii_avarie_p2" : Bool = PLC Avarii.avarie_p2, 1 s
   "Avarii_reset_avarii" : Bool = PLC Avarii.reset_avarii, 1 s
   "Variabile_scara1_start_sus" : Bool = PLC Variabile_scara1.start_sus, 1 s
   "Variabile_scara1_start_jos" : Bool = PLC Variabile_scara1.start_jos, 1 s
   "Variabile_scara2_start_sus" : Bool = PLC Variabile_scara2.start_sus, 1 s
   "Variabile_scara2_start_jos" : Bool = PLC Variabile_scara2.start_jos, 1 s
   "Variabile_poarta1_start_intrare" : Bool = PLC Variabile_poarta1.start_intrare, 1 s
   "Variabile_poarta1_start_iesire" : Bool = PLC Variabile_poarta1.start_iesire, 1 s
   "Variabile_poarta2_start_intrare" : Bool = PLC Variabile_poarta2.start_intrare, 1 s
   "Variabile_poarta2_start_iesire" : Bool = PLC Variabile_poarta2.start_iesire, 1 s
   "Variabile_scara1_senzor_presiune" : Bool = PLC Variabile_scara1.senzor_presiune, 1 s
   "Variabile_scara2_senzor_presiune" : Bool = PLC Variabile_scara2.senzor_presiune, 1 s
   "Variabile_scara2_stop" : Bool = PLC Variabile_scara2.stop, 1 s
   "Variabile_scara1_stop" : Bool = PLC Variabile_scara1.stop, 1 s
   "Variabile_scara1_start" : Bool = PLC Variabile_scara1.start, 1 s
   "Variabile_scara2_start" : Bool = PLC Variabile_scara2.start, 1 s
   "Variabile_poarta2_start" : Bool = PLC Variabile_poarta2.start, 1 s
   "Variabile_poarta1_start" : Bool = PLC Variabile_poarta1.start, 1 s
   "Variabile_poarta1_p_deschis" : Bool = PLC Variabile_poarta1.p_deschis, 1 s
   "Variabile_poarta2_p_deschis" : Bool = PLC Variabile_poarta2.p_deschis, 1 s
   "Variabile_poarta2_alarma" : Bool = PLC Variabile_poarta2.alarma, 1 s
   "Variabile_poarta1_alarma" : Bool = PLC Variabile_poarta1.alarma, 1 s
   "Variabile_poarta1_s1" : Bool = PLC Variabile_poarta1.s1, 1 s
   "Variabile_poarta1_s2" : Bool = PLC Variabile_poarta1.s2, 1 s
   "Variabile_poarta1_stop" : Bool = PLC Variabile_poarta1.stop, 1 s
   "Variabile_poarta1_cartela" : Bool = PLC Variabile_poarta1.cartela, 1 s
   "Variabile_poarta2_s1" : Bool = PLC Variabile_poarta2.s1, 1 s
   "Variabile_poarta2_s2" : Bool = PLC Variabile_poarta2.s2, 1 s
   "Variabile_poarta2_stop" : Bool = PLC Variabile_poarta2.stop, 1 s
   "Variabile_poarta2_cartela" : Bool = PLC Variabile_poarta2.cartela, 1 s
   "Variabile_scara2_curent_triunghi" : Real = PLC Variabile_scara2.curent_triunghi, 1 s
   "Variabile_scara2_curent_stea" : Real = PLC Variabile_scara2.curent_stea, 1 s
   "Variabile_scara1_porniire_stea" : Bool = PLC Variabile_scara1.porniire_stea, 1 s
   "Variabile_scara1_pornire_triunghi" : Bool = PLC Variabile_scara1.pornire_triunghi, 1 s
   "Variabile_scara2_porniire_stea" : Bool = PLC Variabile_scara2.porniire_stea, 1 s
   "Variabile_scara2_pornire_triunghi" : Bool = PLC Variabile_scara2.pornire_triunghi, 1 s
   "Variabile_scara1_cartela_intr" : Bool = PLC Variabile_scara1.cartela_intr, 1 s
   "Variabile_scara2_cartela_intr" : Bool = PLC Variabile_scara2.cartela_intr, 1 s

discrete alarms
   1: 'ESD', class Errors, trigger "Alarme_scara_alarme_gather" bit 0
   2: 'Avarie scara1', class Errors, trigger "Alarme_scara_alarme_gather" bit 1
   3: 'Avarie scara2', class Errors, trigger "Alarme_scara_alarme_gather" bit 2
   4: 'Tensiune necorespunzatoare pe stea 1', class Errors, trigger "Alarme_scara_alarme_gather" bit 3
   5: 'Tensiune necorespunzatoare pe triunghi 1', class Errors, trigger "Alarme_scara_alarme_gather" bit 4
   6: 'Tensiune necorespunzatoare pe stea 2', class Errors, trigger "Alarme_scara_alarme_gather" bit 5
   7: 'Tensiune necorespunzatoare pe triunghi 2', class Errors, trigger "Alarme_scara_alarme_gather" bit 6
   8: 'Avarie poarta 1', class Errors, trigger "Alarme_poarta_alarme_gather" bit 0
   9: 'Avarie poarta 2', class Errors, trigger "Alarme_poarta_alarme_gather" bit 1

Template "Template_1" 800x480
   Button "Exit" at 722,440 size 55x39; TextOff 'Exit'; PictureOff "ExitRuntime_KTP900_Basic_PN_TR"; PictureOn "ExitRuntime_KTP900_Basic_PN_TR"
      on Release: StopRuntime(0)
   Button "Template_Button" at 622,440 size 55x39; TextOff 'Text'
   Button "Template_Button_1" at 522,440 size 55x39; TextOff 'Text'
   Button "Alarms" at 622,440 size 55x39; TextOff 'Alarms'; PictureOff "AlarmDisplay_KTP900_Basic_PN_TR"; PictureOn "AlarmDisplay_KTP900_Basic_PN_TR"
      on Release: function_ef3f5d25("Alarm window_1", -1)
   Button "Start screen" at 522,440 size 55x39; TextOff 'Start screen'; PictureOff "NavigateHome_KTP900_Basic_PN_TR"; PictureOn "NavigateHome_KTP900_Basic_PN_TR"
      on Release: ActivateScreen("Main", 0)
   SymbolicIOField "Symbolic_IO_Field_Screen" at 73,7 size 620x26; TextOff '0'; TextOn '1'; TextList "TextList_ScreenNames"
      ProcessValue <- "Tag_ScreenNumber"
      on Change: ActivateScreenByNumber("Tag_ScreenNumber", 0)
   DateTimeField "HmiScreenItemData" at 695,20 size 105x20
   DateTimeField "HmiScreenItemData_1" at 695,0 size 105x20
   GraphicView "Logo" at 0,0 size 71x40; Picture "Logo of HMI_1"

screen "Main" 800x480, template "Template_1"
   on GenerateScreen: SetTag("Tag_ScreenNumber", 1)
   TextField "Text field_1" at 120,456 size 60x20; Text 'Simulare'
   TextField "Text field_2" at 35,456 size 35x20; Text 'Main'
   TextField "Text field_3" at 683,91 size 43x20; Text 'Avarii'
   Circle "Circle_1" at 646,150 size 34x34
      Appearance <- "Avarii_avarie_s1"
   Button "Button_1" at 705,152 size 72x32; TextOff 'Scara 1'
      on Click: SetBit("Avarii_avarie_s1")
   Circle "Circle_2" at 646,197 size 34x34
      Appearance <- "Avarii_avarie_s2"
   Button "Button_2" at 705,199 size 72x32; TextOff 'Scara 2'
      on Click: SetBit("Avarii_avarie_s2")
   Circle "Circle_3" at 646,244 size 34x34
      Appearance <- "Avarii_avarie_p1"
   Button "Button_3" at 705,246 size 72x32; TextOff 'Poarta 1'
      on Click: SetBit("Avarii_avarie_p1")
   Circle "Circle_4" at 646,291 size 34x34
      Appearance <- "Avarii_avarie_p2"
   Button "Button_4" at 705,293 size 72x32; TextOff 'Poarta 2'
      on Click: SetBit("Avarii_avarie_p2")
   Button "Button_5" at 671,352 size 72x32; TextOff 'Reset'
      on Click: SetBit("Avarii_reset_avarii")
   Circle "Circle_5" at 522,286 size 48x48
      Appearance <- "Avarii_esd"
   Button "Button_6" at 515,343 size 63x32; TextOff 'ESD'
      on Click: SetBit("Avarii_esd_btn")
   Button "Button_7" at 515,386 size 63x32; TextOff 'RESET'
      on Click: SetBit("Avarii_reset_esd")
   TextField "Text field_4" at 39,91 size 54x20; Text 'Scara 1'
   TextField "Text field_5" at 161,92 size 54x20; Text 'Scara 2'
   TextField "Text field_6" at 283,93 size 61x20; Text 'Poarta 1'
   TextField "Text field_7" at 405,94 size 61x20; Text 'Poarta 2'
   IOField "I/O field_1" at 16,146 size 96x32; FormatPattern 9
      ProcessValue <- "Variabile_scara1_curent_triunghi"
   IOField "I/O field_2" at 16,222 size 96x32; FormatPattern 9
      ProcessValue <- "Variabile_scara1_curent_stea"
   TextField "Text field_8" at 47,198 size 35x20; Text 'Stea'
   TextField "Text field_9" at 35,126 size 56x20; Text 'Triunghi'
   IOField "I/O field_3" at 138,146 size 96x32; FormatPattern 9
      ProcessValue <- "Variabile_scara2_curent_triunghi"
   IOField "I/O field_4" at 138,222 size 96x32; FormatPattern 9
      ProcessValue <- "Variabile_scara2_curent_stea"
   Button "Button_12" at 15,330 size 96x32; TextOff 'Jos'
      on Click: SetBit("Variabile_scara1_start_jos")
   Button "Button_13" at 137,330 size 96x32; TextOff 'Jos'
      on Click: SetBit("Variabile_scara2_start_jos")
   Button "Button_14" at 263,330 size 96x32; TextOff 'Iesire'
      on Click: SetBit("Variabile_poarta1_start_iesire")
   Button "Button_15" at 385,330 size 96x32; TextOff 'Iesire'
      on Click: SetBit("Variabile_poarta2_start_iesire")
   Button "Button_16" at 15,285 size 96x32; TextOff 'Sus'
      on Click: SetBit("Variabile_scara1_start_sus")
   Button "Button_17" at 137,285 size 96x32; TextOff 'Sus'
      on Click: SetBit("Variabile_scara2_start_sus")
   Button "Button_18" at 263,285 size 96x32; TextOff 'Intrare'
      on Click: SetBit("Variabile_poarta1_start_intrare")
   Button "Button_19" at 385,285 size 96x32; TextOff 'Intrare'
      on Click: SetBit("Variabile_poarta2_start_intrare")
   TextField "Text field_12" at 167,199 size 35x20; Text 'Stea'
   TextField "Text field_13" at 155,127 size 56x20; Text 'Triunghi'

screen "Simulare" 800x480
   TextField "Text field_1" at 120,456 size 60x20; Text 'Simulare'
   TextField "Text field_2" at 35,456 size 35x20; Text 'Main'
   Rectangle "Rectangle_1" at 55,45 size 83x310
      Appearance <- "Variabile_scara1_start"
   Rectangle "Rectangle_2" at 180,44 size 83x310
      Appearance <- "Variabile_scara2_start"
   TextField "Text field_3" at 71,17 size 54x20; Text 'Scara 1'
   TextField "Text field_4" at 194,17 size 54x20; Text 'Scara 2'
   Button "Button_1" at 64,377 size 61x32; TextOff 'Senzor'
      on Click: SetTag("Variabile_scara1_senzor_presiune", 1)
   Button "Button_2" at 190,375 size 61x32; TextOff 'Senzor'
      on Click: SetTag("Variabile_scara2_senzor_presiune", 1)
   Rectangle "Rectangle_3" at 453,71 size 111x48
      Appearance <- "Variabile_poarta1_start"
   Rectangle "Rectangle_4" at 453,276 size 111x48
      Appearance <- "Variabile_poarta2_start"
   TextField "Text field_5" at 475,36 size 61x20; Text 'Poarta 1'
   TextField "Text field_6" at 475,244 size 61x20; Text 'Poarta 2'
   Button "Button_3" at 63,414 size 61x32; TextOff 'Stop'
      on Click: SetBit("Variabile_scara1_stop")
   Button "Button_4" at 189,412 size 61x32; TextOff 'Stop'
      on Click: SetBit("Variabile_scara2_stop")
   Button "Button_5" at 624,81 size 38x32; TextOff 'S1'
      on Click: SetBit("Variabile_poarta1_s1")
   Button "Button_6" at 682,81 size 38x32; TextOff 'S2'
      on Click: SetBit("Variabile_poarta1_s2")
   Button "Button_7" at 612,128 size 50x32; TextOff 'Stop'
      on Click: SetBit("Variabile_poarta1_stop")
   Button "Button_8" at 682,128 size 50x32; TextOff 'Cartela'
      on Click: SetBit("Variabile_poarta1_cartela")
      Visibility <- "Variabile_poarta1_start_intrare"
   Circle "Circle_1" at 682,174 size 48x48
      Visibility <- "Variabile_poarta1_start_intrare"
      Appearance <- "Variabile_poarta1_alarma"
   TextField "Text field_7" at 614,188 size 51x20; Text 'Alarma'
      Visibility <- "Variabile_poarta1_start_intrare"
   Circle "Circle_2" at 525,146 size 48x48
      Appearance <- "Variabile_poarta1_p_deschis"
   TextField "Text field_8" at 457,160 size 54x20; Text 'Deschis'
   Button "Button_9" at 622,282 size 38x32; TextOff 'S1'
      on Click: SetBit("Variabile_poarta2_s1")
   Button "Button_10" at 680,282 size 38x32; TextOff 'S2'
      on Click: SetBit("Variabile_poarta2_s2")
   Button "Button_11" at 610,333 size 50x32; TextOff 'Stop'
      on Click: SetBit("Variabile_poarta2_stop")
   Button "Button_12" at 680,333 size 50x32; TextOff 'Cartela'
      on Click: SetBit("Variabile_poarta2_cartela")
      Visibility <- "Variabile_poarta2_start_intrare"
   Circle "Circle_3" at 680,375 size 48x48
      Visibility <- "Variabile_poarta2_start_intrare"
      Appearance <- "Variabile_poarta2_alarma"
   TextField "Text field_9" at 612,389 size 51x20; Text 'Alarma'
      Visibility <- "Variabile_poarta2_start_intrare"
   Circle "Circle_4" at 523,347 size 48x48
      Appearance <- "Variabile_poarta2_p_deschis"
   TextField "Text field_10" at 455,361 size 54x20; Text 'Deschis'
   TextField "Text field_11" at 80,144 size 28x20; Text 'Sus'
      Visibility <- "Variabile_scara1_start_sus"
   TextField "Text field_12" at 81,231 size 26x20; Text 'Jos'
      Visibility <- "Variabile_scara1_start_jos"
   TextField "Text field_13" at 204,145 size 28x20; Text 'Sus'
      Visibility <- "Variabile_scara2_start_sus"
   TextField "Text field_14" at 205,232 size 26x20; Text 'Jos'
      Visibility <- "Variabile_scara2_start_jos"
   TextField "Text field_15" at 481,76 size 52x20; Text 'Intrare'
      Visibility <- "Variabile_poarta1_start_intrare"
   TextField "Text field_16" at 487,97 size 42x20; Text 'Iesire'
      Visibility <- "Variabile_poarta1_start_iesire"
   TextField "Text field_17" at 482,279 size 52x20; Text 'Intrare'
      Visibility <- "Variabile_poarta2_start_intrare"
   TextField "Text field_18" at 488,300 size 42x20; Text 'Iesire'
      Visibility <- "Variabile_poarta2_start_iesire"
   Circle "Circle_5" at 290,135 size 27x27
      Appearance <- "Variabile_scara2_porniire_stea"
   TextField "Text field_19" at 286,115 size 35x20; Text 'Stea'
   Circle "Circle_6" at 292,222 size 27x27
      Appearance <- "Variabile_scara2_pornire_triunghi"
   TextField "Text field_20" at 278,202 size 56x20; Text 'Triunghi'
   Circle "Circle_7" at 12,134 size 27x27
      Appearance <- "Variabile_scara1_porniire_stea"
   TextField "Text field_21" at 8,114 size 35x20; Text 'Stea'
   Circle "Circle_8" at 14,221 size 27x27
      Appearance <- "Variabile_scara1_pornire_triunghi"
   TextField "Text field_22" at 0,201 size 56x20; Text 'Triunghi'
   Circle "Circle_9" at 743,131 size 27x27
      Appearance <- "Variabile_scara1_cartela_intr"
      Visibility <- "Variabile_poarta1_start_intrare"
   Circle "Circle_10" at 742,335 size 27x27
      Appearance <- "Variabile_scara2_cartela_intr"
      Visibility <- "Variabile_poarta2_start_intrare"
   Button "Button_13" at 260,376 size 24x32; TextOff 'R'
      on Click: SetTag("Variabile_scara2_senzor_presiune", 0)
   Button "Button_14" at 33,376 size 24x32; TextOff 'R'
      on Click: SetTag("Variabile_scara1_senzor_presiune", 0)
*)